FUNCTION ScalingOut : BOOL
VAR_INPUT
END_VAR
VAR
	HoistingScaling: INT := 300;
	PumpScaling: INT := 100;
	IntMax : INT := 32767;
END_VAR

//Allows no motor movement when either door is open
IF (Inputs.DOORSENS1 = FALSE OR Inputs.DOORSENS2 = FALSE) THEN
	Outputs.AO_HOISTING := 0;
	RETURN;
END_IF

// Prevent integer overflow which causes motor to run in reverse
IF Process.HoistingDemandValue >= HoistingScaling THEN
	Process.HoistingDemandValue := INT_TO_REAL(HoistingScaling);
ELSIF Process.HoistingDemandValue <= (-1) * HoistingScaling THEN
	Process.HoistingDemandValue:= INT_TO_REAL(HoistingScaling*(-1));
END_IF

//Prevent integer overflow and sub-zero values
IF Process.PumpPID >= PumpScaling THEN
	Process.PumpPID := REAL_TO_INT(PumpScaling);
ELSIF Process.PumpPID <= 0 THEN
	Process.PumpPID := 0;
END_IF


//Only downwards when top switch is pressed
IF (Inputs.DI_HOISTING_LIM_TOP = FALSE) AND (Process.HoistingDemandValue > 0) THEN
	Outputs.AO_HOISTING := 0;
//Only upwards when bottom switch is pressed
ELSIF (Inputs.DI_HOISTING_LIM_BOTTOM = FALSE) AND (Process.HoistingDemandValue < 0) THEN
	Outputs.AO_HOISTING := 0;
ELSE
	Outputs.AO_HOISTING := REAL_TO_INT(Process.HoistingDemandValue/HoistingScaling*IntMax);
END_IF

Outputs.AO_ValveWaterIn := DINT_TO_INT(Process.PumpOpen*IntMax);

Outputs.DO_PumpEnable := DINT_TO_BOOL(Process.PumpEnable);
Outputs.AO_PUMP := REAL_TO_INT(Process.PumpPID/PumpScaling*IntMax);

END_FUNCTION

(* stored: Version 1.1.0.1, ProductVersion 3.1.4024.9
   POU ScalingOut: Id {5d485be6-0ae8-49f7-9e70-8e9a4220cc67}, SpecialFunc None *)
